// TwinCAT 3 PLC project Untitled1
// ProgramVersion: 3.1.4024.0
// libraries:
//   Tc2_Standard, * (Beckhoff Automation GmbH)
//   Tc2_System, * (Beckhoff Automation GmbH)
//   Tc3_Module, * (Beckhoff Automation GmbH)
// project tree:
//   FB/ FB_ST10.TcPOU, FB_ST10b.TcPOU
//   / PlcTask.TcTTO
//   POUs/ MAIN.TcPOU
// real-time tasks:
//   TASK PlcTask: cycle T#10ms, priority 20, ADS port 350

CONFIGURATION Untitled1
    RESOURCE PLC ON TwinCAT3
        TASK PlcTask(INTERVAL := T#10ms, PRIORITY := 20);
        PROGRAM MAIN WITH PlcTask : MAIN;
    END_RESOURCE
END_CONFIGURATION

// ---- POUs/MAIN.TcPOU
PROGRAM MAIN
VAR
	_fb : FB_ST10; 
	_test : BOOL;
END_VAR

IF _fb._robot() THEN 
	_test:= TRUE; 
ELSE 
	_test:= FALSE; 
END_IF
_fb._tcpIp();
IF _fb._scanner() THEN 
	_test:= FALSE; 
END_IF

END_PROGRAM

// ---- FB/FB_ST10.TcPOU
FUNCTION_BLOCK FB_ST10
VAR
	_camera : BOOL;
	_triger : BOOL;
	_description : STRING;
	_test : BOOL;
	_cameraProgram : UINT;
	_gitTest : BOOL;
	_git : INT;
	_ivana : INT;
	_var : INT; 
	_i : INT; 
	
END_VAR

METHOD PROTECTED _camera
VAR_INPUT
END_VAR
IF _camera THEN 
	_description:= 'On';
	_cameraProgram:= 1;
ELSE 
	_cameraProgram:= 5; 
	_triger:= TRUE; 
END_IF

_var:= 55;
END_METHOD

METHOD _robot : BOOL
VAR_INPUT
END_VAR
END_METHOD

METHOD _scanner : BOOL
VAR_INPUT
END_VAR
IF _triger THEN 
	_description:= 'Trger scanner';
END_IF
_gitTest:= TRUE; 
_ivana := 5;
END_METHOD

METHOD _tcpIp
VAR_INPUT
END_VAR
_test:= TRUE; 
_ivana:= 5;
END_METHOD

METHOD _test : BOOL
VAR_INPUT
END_VAR
END_METHOD

END_FUNCTION_BLOCK

// ---- FB/FB_ST10b.TcPOU
FUNCTION_BLOCK FB_ST10b
VAR
	_test : BOOL; 
END_VAR

METHOD _test : BOOL
VAR_INPUT
END_VAR
_test:= TRUE;
END_METHOD

END_FUNCTION_BLOCK
